Universal Robots PolyScope program: test_base_bridgeD.urp

Program test_base_bridgeD (installation=default directory=/ursim/programs createdIn=3.2.19275 lastSavedIn=5.19.0 robotSerialNumber=20195599999)
Calibrated DH parameters: a=[0, -0.425, -0.3922, 0, 0, 0]; d=[0.1625, 0, 0, 0.1333, 0.0997, 0.0996]; alpha=[1.570796, 0, 0, 1.570796, -1.570796, 0]; deltaTheta=[0, 0, 0, 0, 0, 0]
InitVariablesNode
BeforeStart
  syncPos := p[0,1.6,2.25,0,1.57,0]
  Script file /ursim/programs/addFunctons.script
    | global p=0
    | global theta = 1.57
    | global r = 0.1
    | global f = 0.2
    | 
    | global syncPos = p[0.452,0.13834,0.6810,2.389,-2.494,2.141]
    | def cPose(p,theta,r,f):
    |     p = p + f*(2*3.1415/500)
    |     z = r*sin(theta + p )
    |     y = r*cos(theta + p )
    | return [y,z,p]
    | 
    | end
    | def addTrackedTcp(x,y,z):
    |     x = tcpPartner[0] + x
    |     y = tcpPartner[1] + y
    |     z = tcpPartner[2] + z
    | return [x,y,z]
    | end
    | 
    | def addTrackedTcp2(x,y,z):
    |     mypose =  get_actual_tcp_pose()
    |     x = mypose[0] + x
    |     y = mypose[1] + y
    |     z = mypose[2] + z
    |     global original_tpc = mypose
    | return [x,y,z,mypose[3],mypose[4],mypose[5]]
    | end
    | 
    | def moveNext():
    |     pos_p = cPose(p,theta,r,f)
    |     # popup(pos_p,"c pose",blocking = True)
    |     p = pos_p[2]
    |     global nextPosition = addTrackedTcp(0,pos_p[0], pos_p[1])
    |     # popup(nextPosition,"position",blocking = False)
    |     q = get_inverse_kin(p[nextPosition[0],nextPosition[1],nextPosition[2],tcpPartner[3],tcpPartner[4],tcpPartner[5]])
    |     servoj(q,0.5,500)
    | end
    | 
    | def moveFromAtoB(center):
    |     pointA = center
    |     pointB = center
    |     pointA[1] = pointA[1] + 0.4
    |     pointB[1] = pointB[1] - 0.4
    |     movel(pointA,v = 0.130)
    |     movel(pointB)
    | end
    | def movejOffset(point,x,y,z):
    |     point[0] = point[0] + x
    |     point[1] = point[1] + y
    |     point[2] = point[2] + z
    |     movej(point)
    | end
  Script file /ursim/programs/bridgeBeforeStart.script
    | global tcpPartner = p[0, 0, 0, 0, 0, 0]
    | global ftPartner = p[0, 0, 0, 0, 0, 0]
    | global inPosSync = 1
    | global go = 0
    | write_output_integer_register(24, 0)
    | 
    | while (inPosSync != 0):
    |     global inPosSync = read_input_integer_register(24)
    | end
    | 
    | popup("entered","entered")
    | movej(syncPos, a=1.3962634015954636, v=1.0471975511965976)
    | write_output_integer_register(24, 1)
    | 
    | while (inPosSync != 1):
    |     global inPosSync = read_input_integer_register(24)
    | end
    | 
    | sleep(0.1)
Robot Program (runOnlyOnce=false)
  SuppressedNode
    Script: startTime = time(mode = 2)
  go := read_input_integer_register(24)
  SuppressedNode
    MoveJ speed 60 deg/s, acceleration 80 deg/s^2 (useActiveTCP=true) feature=Base
      Waypoint Variable (Variable): variable=syncPos
  Script: movejOffset(syncPos,0,0,0.20)
  Script: write_output_integer_register(24, 2)
  SuppressedNode
    go := 2
  If go ≟2
    Loop Forever
      Script: moveNext()
Thread Thread_1 (runOnlyOnce=false)
  Loop Forever
    tmpTcp := p[0,0,0,0,0,0]
    Script: tmpTcp[0] = read_input_float_register(24)
    Script: tmpTcp[1] = read_input_float_register(25)
    Script: tmpTcp[2] = read_input_float_register(26)
    Script: tmpTcp[3] = read_input_float_register(27)
    Script: tmpTcp[4] = read_input_float_register(28)
    Script: tmpTcp[5] = read_input_float_register(29)
    tcpPartner := tmpTcp
    Script: sync()
Thread Thread_2 (runOnlyOnce=false)
  Loop Forever
    tmp := p[0,0,0,0,0,0]
    Script: tmp[0] = read_input_float_register(30)
    Script: tmp[1] = read_input_float_register(31)
    Script: tmp[2] = read_input_float_register(32)
    Script: tmp[3] = read_input_float_register(33)
    Script: tmp[4] = read_input_float_register(34)
    Script: tmp[5] = read_input_float_register(35)
    ftPartner := tmp
    Script: sync()
